// TIA Portal V19 export
DATA_BLOCK "ControlDB"   // DB3
{ S7_Optimized_Access := 'TRUE' }
// stored: MemoryReserve 100
   VAR
      CanProcessImageIn : Array[0..31] of Byte;
      CanProcessImageOut : Array[0..9] of Byte;
      ReadCanProcessImageBusy : Bool;
      ReadCanProcessImageError : Bool;
      ReadCanProcessImageSize : UInt;
      ReadCanProcessImageStatus : DWord;
      ReadCanProcessImageValid : Bool;
      WriteCanProcessImageBusy : Bool;
      WriteCanProcessImageError : Bool;
      WriteCanProcessImageSize : UInt;
      WriteCanProcessImageStatus : DWord;
      WriteCanProcessImageDone : Bool;
      ErrorRegisterReq : Bool;
      ErrorRegisterNode : Int;
      ErrorRegisterBusy : Bool;
      ErrorRegisterGenericError : Bool;
      ErrorRegisterCurrentError : Bool;
      ErrorRegisterVoltageError : Bool;
      ErrorRegisterTemperatureError : Bool;
      ErrorRegisterCommunicationError : Bool;
      ErrorRegisterDeviceSpecificError : Bool;
      ErrorRegisterManufacturerSpecificError : Bool;
      HeartbeatReq : Bool;
      HeartbeatNode : Int;
      HeartbeatMilliseconds : UInt;
      HeartbeatBusy : Bool;
   END_VAR
BEGIN
   CanProcessImageOut[0] := 16#F0;
END_DATA_BLOCK
